PROGRAM MAIN
VAR
END_VAR

Reaktoranlage();

END_PROGRAM

(* stored: Version 1.1.0.1, ProductVersion 3.1.4024.12
   POU MAIN: Id {26b9df25-7643-42fb-8a0d-7af5b34d4ed3}, SpecialFunc None *)
